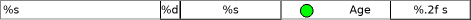
VISUALIZATION VISU_AlpacaGetCoverState  // 471x20
VAR_IN_OUT
	stInstance : ST_AlpacaGetCoverState;
END_VAR
    Rectangle (160,0 20x20), "%d", text variable: stInstance.nValue
    Rectangle (0,0 161x20), "%s", text variable: stInstance.sName
    Ellipse (300,4 13x13), colour toggle: stInstance.eStatusCode <> E_AlpacaStatusCode.OK
    Rectangle (390,0 81x20), "%.2f s", text variable: stInstance.rAge
    Label (340,0 41x20), "Age"
    Rectangle (180,0 101x20), "%s", text variable: stInstance.sValue
END_VISUALIZATION

(* stored: Version 1.1.0.1, ProductVersion 3.1.4024.12
   Visu VISU_AlpacaGetCoverState: Id {40ca58a5-fd5a-4a2b-98c9-3bddbc2a29f0} *)
